{attribute 'pack_mode' := '1'}
TYPE ST_TcpTask2 :
STRUCT
	TaskName : STRING(24);
	TaskType : INT; (* 0:Once, 1:Regular *)
	pData : PVOID;
	nData : UDINT;
END_STRUCT
END_TYPE

(* stored: Version 1.1.0.1, ProductVersion 3.1.4024.12
   DUT ST_TcpTask2: Id {812356c4-5d83-43af-b11d-7001142b415f} *)
